PROGRAM MAIN
VAR
	fbMotor : FB_Motor;
    fbValve : FB_Valve;

    tMotorFB : TON;
	tValveOpenFB : TON;
	tValveCloseFB : TON;

    rtPiece : R_TRIG;
    tDelay  : TON;
    tBlow   : TON;

    MachineState : State_Machine := ST_IDLE;
END_VAR

rtPiece(CLK := PieceSensor);

fbMotor.Start := FALSE;
fbMotor.Stop := FALSE;
fbValve.OpenCmd := FALSE;
fbValve.CloseCmd := FALSE;

CASE MachineState OF

ST_IDLE:
    fbMotor.Start := FALSE;

    IF Start THEN
        MachineState := ST_RUN;
    END_IF


ST_RUN:

    fbMotor.Start := TRUE;
    fbMotor.Stop := FALSE;

    IF rtPiece.Q THEN
        tDelay(IN := TRUE, PT := T#500ms);
    ELSE
        tDelay(IN := FALSE);
    END_IF

    IF tDelay.Q THEN
        tBlow(IN := TRUE, PT := T#300ms);
    ELSE
        tBlow(IN := FALSE);
    END_IF

    fbValve.OpenCmd := tBlow.IN;
    fbValve.CloseCmd := tBlow.Q;

    // ERRORI
    IF fbMotor.Fault OR fbValve.Fault THEN
        MachineState := ST_ERROR;
    END_IF

    IF Stop THEN
        MachineState := ST_IDLE;
    END_IF


ST_ERROR:

    fbMotor.Start := FALSE;
    fbValve.OpenCmd := FALSE;
    fbValve.CloseCmd := FALSE;

    IF Reset THEN
        MachineState := ST_IDLE;
    END_IF

END_CASE

fbMotor(
    MotorFeedback := SimMotorFB,
    EStop := EStop,
    InterlockOK := InterlockOK,
    Reset := Reset
);

fbValve(
    OpenFeedback := SimOpenFB,
    CloseFeedback := SimCloseFB,
    E_Stop := EStop,
    InterlockOK := InterlockOK,
    Reset := Reset
);

// SIMULAZIONE FEEDBACK

// Motor feedback
IF fbMotor.MotorCmd THEN
    tMotorFB(IN := TRUE, PT := T#1s);
ELSE
    tMotorFB(IN := FALSE);
END_IF;
SimMotorFB := tMotorFB.Q;

// Open feedback
IF fbValve.OpenOut THEN
    tValveOpenFB(IN := TRUE, PT := T#3S);
ELSE
    tValveOpenFB(IN := FALSE);
END_IF;

// Close feedback
IF fbValve.CloseOut THEN
    tValveCloseFB(IN := TRUE, PT := T#10S);
ELSE
    tValveCloseFB(IN := FALSE);
END_IF;
SimOpenFB := tValveOpenFB.Q;
SimCloseFB := tValveCloseFB.Q;

// Mapping Output
MotorOut     := fbMotor.MotorCmd;
ValveOpenOut := fbValve.OpenOut;
ValveCloseOut := fbValve.CloseOut;

END_PROGRAM

(* stored: Version 1.1.0.1, ProductVersion 3.1.4024.16
   POU MAIN: Id {d862376b-c84c-4576-a80c-631cfd95d38c}, SpecialFunc None *)
